// Mitsubishi GX Works2 project: PLC_GROUP13   PLC: FX3G

// global labels: Global1
VAR_GLOBAL
  StartDay AT X007 : BOOL;
END_VAR
VAR_GLOBAL CONSTANT
  input_choc : REAL := 1200;
END_VAR
VAR_GLOBAL
  chocStock AT D1152 : REAL;
END_VAR
VAR_GLOBAL CONSTANT
  input_nuts : REAL := 300;
END_VAR
VAR_GLOBAL
  nutsStock AT D1156 : REAL;
END_VAR
VAR_GLOBAL CONSTANT
  input_pist : REAL := 300;
END_VAR
VAR_GLOBAL
  pistStock AT D1160 : REAL;
END_VAR
VAR_GLOBAL CONSTANT
  input_kad : REAL := 120;
END_VAR
VAR_GLOBAL
  kadStock AT D1164 : REAL;
  melt AT X001 : BOOL;
END_VAR
VAR_GLOBAL CONSTANT
  subChoc : REAL := 400;
END_VAR
VAR_GLOBAL
  meltPot AT D1166 : REAL;
END_VAR
VAR_GLOBAL CONSTANT
  meltAdd : REAL := 400;
END_VAR
VAR_GLOBAL
  meltingIndicator AT Y001 : BOOL;
  fillStock AT M7 : BOOL;
END_VAR
VAR_GLOBAL CONSTANT
  minChoc : REAL := 400;
  minNuts : REAL := 100;
  minPist : REAL := 120;
  minKad : REAL := 60;
END_VAR
VAR_GLOBAL
  startDayLamp AT Y007 : BOOL;
END_VAR
VAR_GLOBAL CONSTANT
  Degrees : INT := 45;
END_VAR
VAR_GLOBAL
  TC_0 AT TC0 : BOOL;
  TC_1 AT TC1 : BOOL;
  TS_1 AT TS1 : BOOL;
  meltingProcess AT Y001 : BOOL;
  meltingEnded AT M3 : BOOL;
END_VAR
VAR_GLOBAL CONSTANT
  fourTrays : INT := 4;
END_VAR
VAR_GLOBAL
  placeTrays AT CC3 : BOOL;
  enterTray AT X010 : BOOL;
  traysPlaced AT CS3 : BOOL;
END_VAR
VAR_GLOBAL CONSTANT
  meltePour : REAL := 400;
  fourSeconds : INT := 40;
END_VAR
VAR_GLOBAL
  TC_2 AT TC2 : BOOL;
  pouring AT TC3 : BOOL;
  pouringEnded AT M4 : BOOL;
  pourChoc AT TS3 : BOOL;
  hi AT TS3 : BOOL;
  pourProcess AT Y002 : BOOL;
END_VAR
VAR_GLOBAL CONSTANT
  meltedPour : REAL := 400;
END_VAR
VAR_GLOBAL
  meltedChocPoured AT M6 : BOOL;
  chocMoved AT M5 : BOOL;
  meltingTime AT TC2 : BOOL;
  meltedPoured AT M6 : BOOL;
  applyChocType AT X004 : BOOL;
  chocTypeInput AT D8280 : INT;
  chocTypeSelected AT M10 : BOOL;
END_VAR
VAR_GLOBAL CONSTANT
  minForNuts : REAL;
  maxForNuts : REAL := 2025;
  minForDubai : REAL := 2025;
  maxForDubai : REAL := 4030;
  notGood : REAL := 3920;
  chocTypeNum : REAL := 1;
  removeNutsForNuts : REAL := 100;
  removePistForNuts : REAL := 100;
  nutsForFill : REAL := 200;
END_VAR
VAR_GLOBAL
  nutsMixing AT D1168 : REAL;
END_VAR
VAR_GLOBAL CONSTANT
  fillForNuts : REAL := 200;
  removeNutsForDubai : REAL := 20;
  removePistForDubai : REAL := 120;
  removeKadForDubai : REAL := 60;
  fillForDubai : REAL := 200;
END_VAR
VAR_GLOBAL
  dubaiMixing AT D1170 : REAL;
  mixingPot AT D1168 : REAL;
  ingredientsPoured AT M8 : BOOL;
  flashingLamp AT M9 : BOOL;
END_VAR
VAR_GLOBAL CONSTANT
  flashing3 : REAL := 50;
  fiveSec : INT := 50;
END_VAR
VAR_GLOBAL
  lampY3 AT Y003 : BOOL;
  lampY4 AT Y004 : BOOL;
  wordToReal AT M10 : BOOL;
  chocType1 AT D8202 : REAL;
  chocSelected AT M11 : BOOL;
  flashingTimerFive AT TC6 : BOOL;
  flashTimerEnd AT TS6 : BOOL;
  finishFlashingIndicator AT M12 : BOOL;
  chocSelection AT D1172 : REAL;
END_VAR
VAR_GLOBAL CONSTANT
  nutsSelected1 : REAL := 1;
  dubaiBling : REAL := 2;
  dubaiBling1 : REAL := 2;
END_VAR
VAR_GLOBAL
  chocIdentified AT M13 : BOOL;
  m_20 AT M20 : BOOL;
  m_21 AT M21 : BOOL;
END_VAR
VAR_GLOBAL CONSTANT
  fillForNuts1 : REAL := 200;
END_VAR
VAR_GLOBAL
  w AT M30 : BOOL;
END_VAR
VAR_GLOBAL CONSTANT
  halfSec : INT := 5;
END_VAR
VAR_GLOBAL
  coolChoc AT X006 : BOOL;
  TC_6 AT TC6 : BOOL;
  TS_6 AT TS6 : BOOL;
  coolingLamp AT Y006 : BOOL;
  finishCoolingIndicator AT M13 : BOOL;
  packTray AT X000 : BOOL;
  Packing AT CC4 : BOOL;
  traysPacked AT D1174 : REAL;
END_VAR
VAR_GLOBAL CONSTANT
  oneTray : REAL := 1;
  threeSeconds : INT := 30;
END_VAR
VAR_GLOBAL
  TS_7 AT TS7 : BOOL;
  PackingStartedIndicator AT M14 : BOOL;
  fourTraysPacked AT D1176 : REAL;
END_VAR
VAR_GLOBAL CONSTANT
  onePack : REAL := 1;
END_VAR
VAR_GLOBAL
  iterationEnded AT M15 : BOOL;
  emergency AT X005 : BOOL;
END_VAR
VAR_GLOBAL CONSTANT
  DivideByTen : REAL := 10;
END_VAR
VAR_GLOBAL
  trayscountOutput AT D8282 : INT;
END_VAR
VAR_GLOBAL CONSTANT
  zeroValue : REAL;
END_VAR
VAR_GLOBAL
  emergencyLamp AT M16 : BOOL;
END_VAR
VAR_GLOBAL CONSTANT
  fiftynine : REAL := 59;
END_VAR
VAR_GLOBAL
  outofStockLamp AT M17 : BOOL;
  intkadstock AT D1178 : INT;
  output AT D8282 : INT;
END_VAR
VAR_GLOBAL CONSTANT
  fourhundred : INT := 400;
  fourTy : REAL := 40;
  zero : INT;
END_VAR
VAR_GLOBAL
  dontaddLamp AT M18 : BOOL;
END_VAR
VAR_GLOBAL CONSTANT
  false_0 : BOOL;
END_VAR
VAR_GLOBAL
  meltingTimerFinished AT TS2 : BOOL;
  SelectedNuts AT M20 : BOOL;
  SelectedDubai AT M21 : BOOL;
  flashingTimer4 AT TC4 : BOOL;
  flashingTimer5 AT TC5 : BOOL;
  flashing4finish AT TS4 : BOOL;
  flashing5finish AT TS5 : BOOL;
  coolingTimer AT TC7 : BOOL;
  coolingTimerFinish AT TS7 : BOOL;
  Packed4Trays AT CS4 : BOOL;
  packingLamp AT Y005 : BOOL;
  chocInput AT D1180 : REAL;
  nutsInput AT D1182 : REAL;
  pistInput AT D1184 : REAL;
  kadInput AT D1186 : REAL;
END_VAR

// task Task_01 (event TRUE, interval 0, priority 31): POU_01

PROGRAM POU_01
VAR CONSTANT
  threeSec : INT := 30;
END_VAR
(* structured ladder/FBD written out as ST: instructions are called as NAME(EN, inputs, outputs); _pN, _eN, _tN stand for wires *)
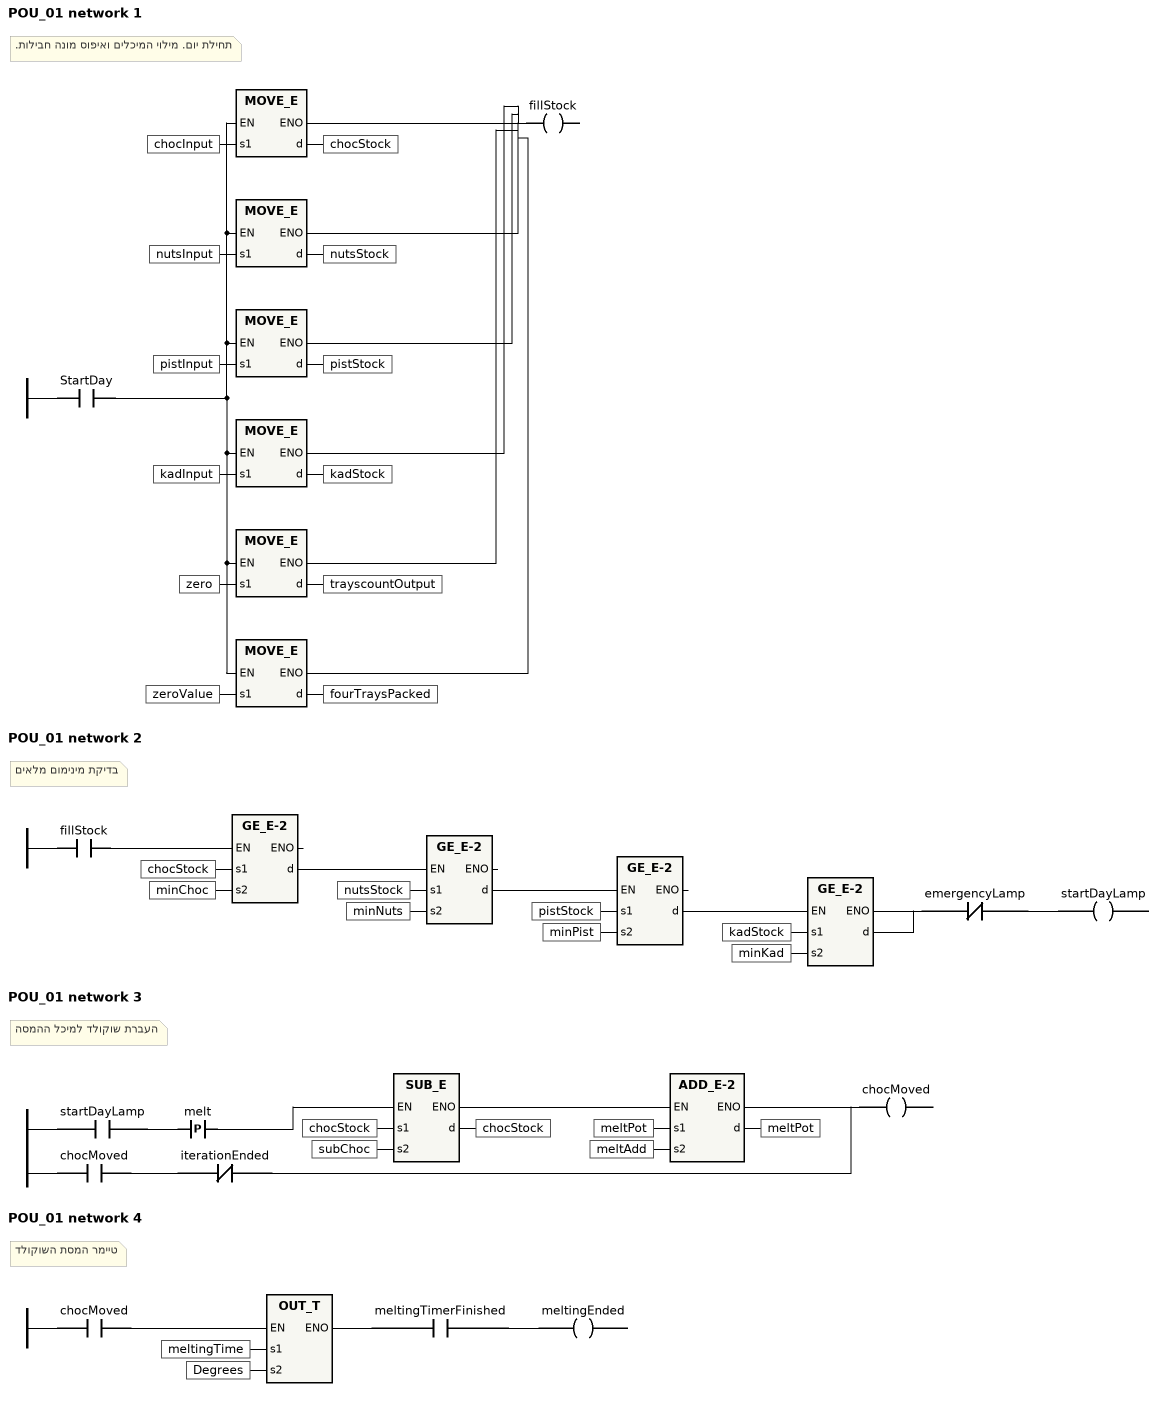
(* network 1 *)
(* תחילת יום. מילוי המיכלים ואיפוס מונה חבילות. *)
_e1 := MOVE_E(StartDay, chocInput, chocStock);
_e2 := MOVE_E(StartDay, nutsInput, nutsStock);
_e3 := MOVE_E(StartDay, pistInput, pistStock);
_e4 := MOVE_E(StartDay, kadInput, kadStock);
_e5 := MOVE_E(StartDay, zero, trayscountOutput);
_e6 := MOVE_E(StartDay, zeroValue, fourTraysPacked);
fillStock := _e1 OR _e2 OR _e3 OR _e4 OR _e5 OR _e6;
(* network 2 *)
(* בדיקת מינימום מלאים *)
GE_E(fillStock, chocStock, minChoc, _t1);
GE_E(_t1, nutsStock, minNuts, _t2);
GE_E(_t2, pistStock, minPist, _t3);
_e5 := GE_E(_t3, kadStock, minKad, _t4);
startDayLamp := (_e5 OR _t4) AND NOT emergencyLamp;
(* network 3 *)
(* העברת שוקולד למיכל ההמסה *)
_e1 := SUB_E(startDayLamp AND LDP(TRUE, melt), chocStock, subChoc, chocStock);
_e2 := ADD_E(_e1, meltPot, meltAdd, meltPot);
chocMoved := _e2 OR (chocMoved AND NOT iterationEnded);
(* network 4 *)
(* טיימר המסת השוקולד *)
_e1 := OUT_T(chocMoved, meltingTime, Degrees);
meltingEnded := _e1 AND meltingTimerFinished;
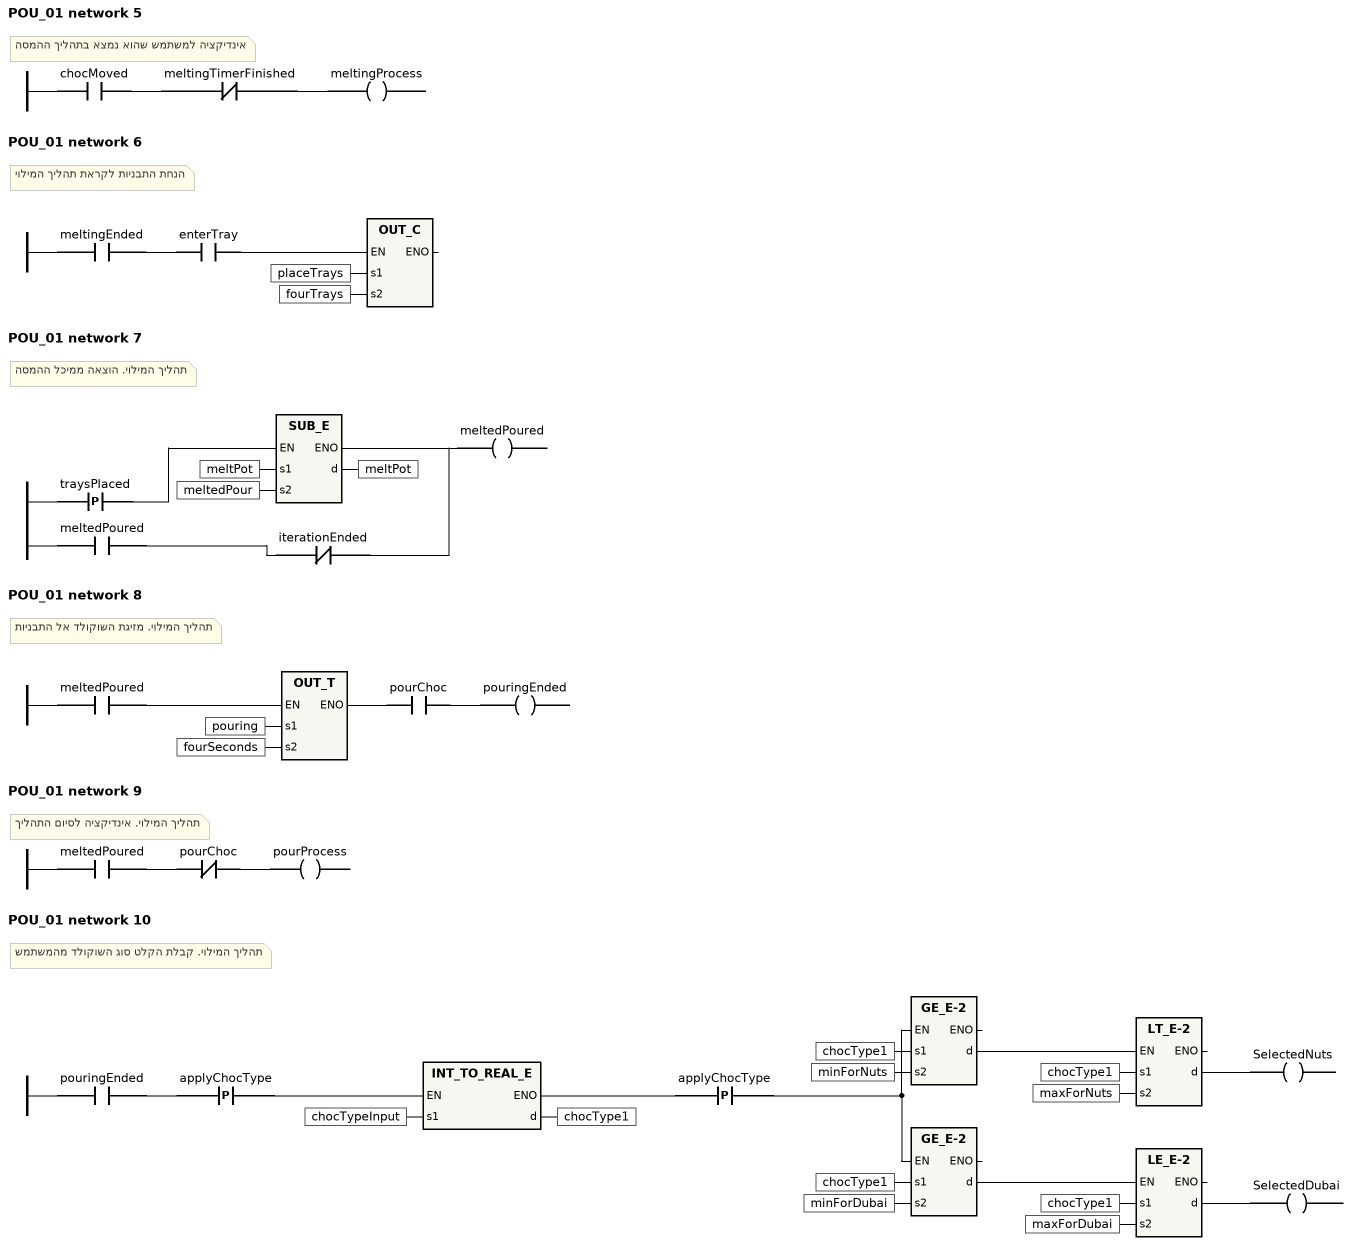
(* network 5 *)
(* אינדיקציה למשתמש שהוא נמצא בתהליך ההמסה *)
meltingProcess := chocMoved AND NOT meltingTimerFinished;
(* network 6 *)
(* הנחת התבניות לקראת תהליך המילוי *)
OUT_C(meltingEnded AND enterTray, placeTrays, fourTrays);
(* network 7 *)
(* תהליך המילוי. הוצאה ממיכל ההמסה *)
_e1 := SUB_E(LDP(TRUE, traysPlaced), meltPot, meltedPour, meltPot);
meltedPoured := _e1 OR (meltedPoured AND NOT iterationEnded);
(* network 8 *)
(* תהליך המילוי. מזיגת השוקולד אל התבניות *)
_e1 := OUT_T(meltedPoured, pouring, fourSeconds);
pouringEnded := _e1 AND pourChoc;
(* network 9 *)
(* תהליך המילוי. אינדיקציה לסיום התהליך *)
pourProcess := meltedPoured AND NOT pourChoc;
(* network 10 *)
(* תהליך המילוי. קבלת הקלט סוג השוקולד מהמשתמש *)
_e1 := INT_TO_REAL_E(pouringEnded AND LDP(TRUE, applyChocType), chocTypeInput, chocType1);
_p2 := _e1 AND LDP(TRUE, applyChocType);
GE_E(_p2, chocType1, minForNuts, _t3);
LT_E(_t3, chocType1, maxForNuts, _t4);
SelectedNuts := _t4;
GE_E(_p2, chocType1, minForDubai, _t5);
LE_E(_t5, chocType1, maxForDubai, _t6);
SelectedDubai := _t6;
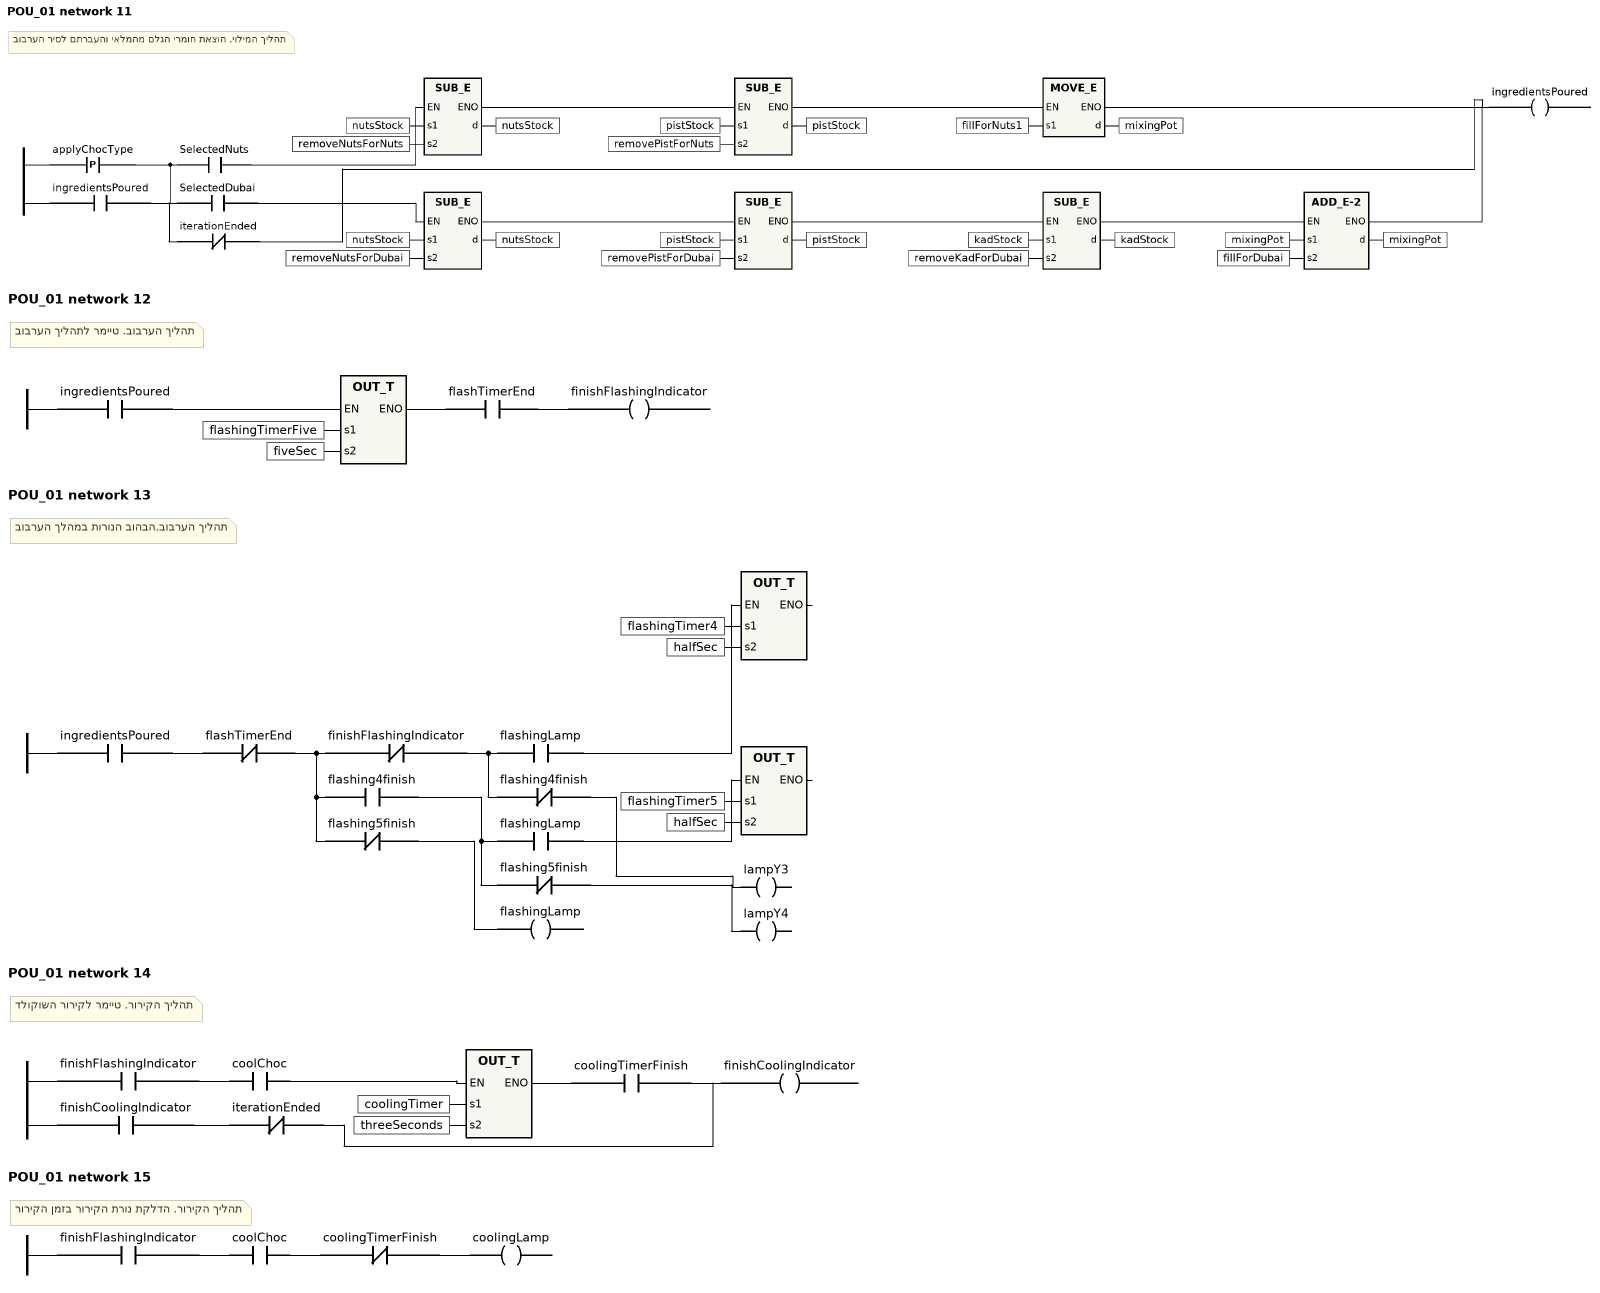
(* network 11 *)
(* תהליך המילוי. הוצאת חומרי הגלם מהמלאי והעברתם לסיר הערבוב *)
_p1 := LDP(TRUE, applyChocType);
_e2 := SUB_E(_p1 AND SelectedNuts, nutsStock, removeNutsForNuts, nutsStock);
_e3 := SUB_E(_e2, pistStock, removePistForNuts, pistStock);
_e4 := MOVE_E(_e3, fillForNuts1, mixingPot);
_e5 := SUB_E(_p1 AND SelectedDubai, nutsStock, removeNutsForDubai, nutsStock);
_e6 := SUB_E(_e5, pistStock, removePistForDubai, pistStock);
_e7 := SUB_E(_e6, kadStock, removeKadForDubai, kadStock);
_e8 := ADD_E(_e7, mixingPot, fillForDubai, mixingPot);
ingredientsPoured := _e4 OR _e8 OR (ingredientsPoured AND NOT iterationEnded);
(* network 12 *)
(* תהליך הערבוב. טיימר לתהליך הערבוב *)
_e1 := OUT_T(ingredientsPoured, flashingTimerFive, fiveSec);
finishFlashingIndicator := _e1 AND flashTimerEnd;
(* network 13 *)
(* תהליך הערבוב.הבהוב הנורות במהלך הערבוב *)
_p1 := ingredientsPoured AND NOT flashTimerEnd;
_p2 := _p1 AND NOT finishFlashingIndicator;
OUT_T(_p2 AND flashingLamp, flashingTimer4, halfSec);
lampY3 := _p2 AND NOT flashing4finish;
_p3 := _p1 AND flashing4finish;
OUT_T(_p3 AND flashingLamp, flashingTimer5, halfSec);
lampY4 := _p3 AND NOT flashing5finish;
flashingLamp := _p1 AND NOT flashing5finish;
(* network 14 *)
(* תהליך הקירור. טיימר לקירור השוקולד *)
_e1 := OUT_T(finishFlashingIndicator AND coolChoc, coolingTimer, threeSeconds);
finishCoolingIndicator := (_e1 AND coolingTimerFinish) OR (finishCoolingIndicator AND NOT iterationEnded);
(* network 15 *)
(* תהליך הקירור. הדלקת נורת הקירור בזמן הקירור *)
coolingLamp := finishFlashingIndicator AND coolChoc AND NOT coolingTimerFinish;
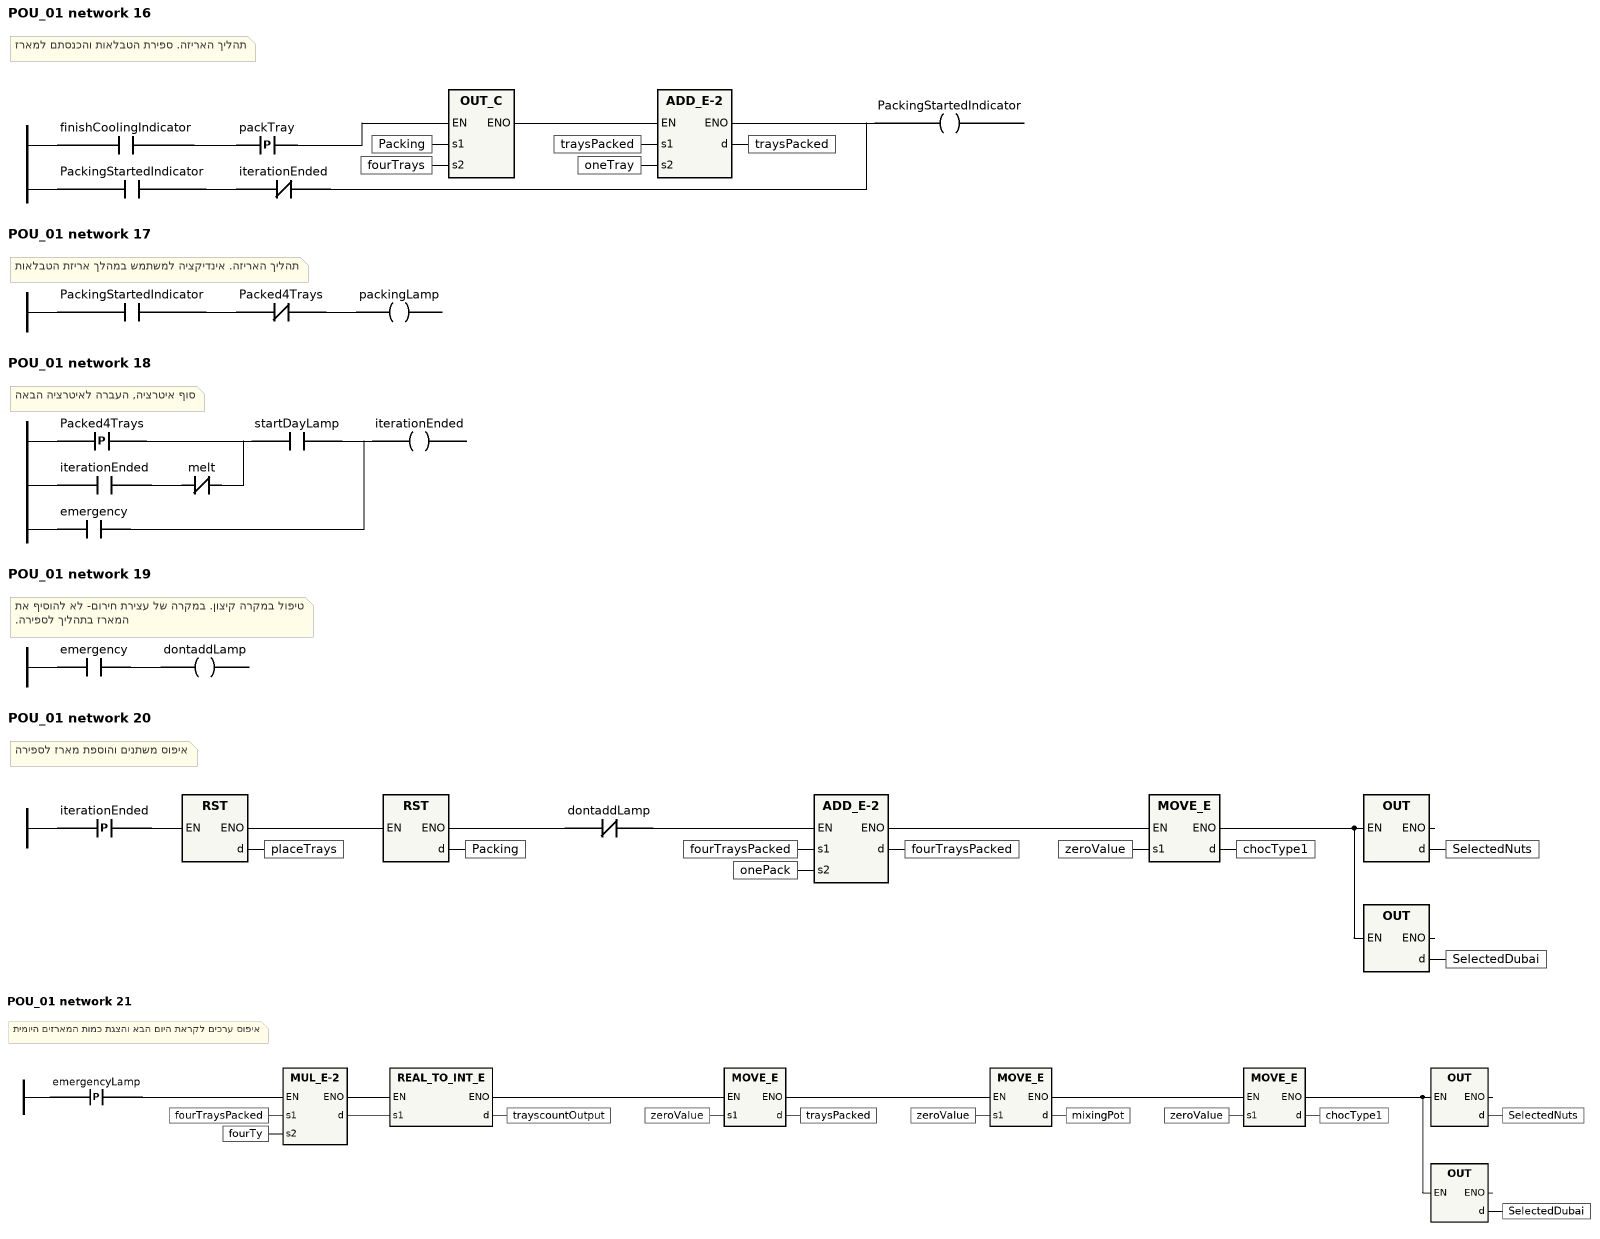
(* network 16 *)
(* תהליך האריזה. ספירת הטבלאות והכנסתם למארז *)
_e1 := OUT_C(finishCoolingIndicator AND LDP(TRUE, packTray), Packing, fourTrays);
_e2 := ADD_E(_e1, traysPacked, oneTray, traysPacked);
PackingStartedIndicator := _e2 OR (PackingStartedIndicator AND NOT iterationEnded);
(* network 17 *)
(* תהליך האריזה. אינדיקציה למשתמש במהלך אריזת הטבלאות *)
packingLamp := PackingStartedIndicator AND NOT Packed4Trays;
(* network 18 *)
(* סוף איטרציה, העברה לאיטרציה הבאה *)
iterationEnded := ((LDP(TRUE, Packed4Trays) OR (iterationEnded AND NOT melt)) AND startDayLamp) OR emergency;
(* network 19 *)
(* טיפול במקרה קיצון. במקרה של עצירת חירום- לא להוסיף את המארז בתהליך לספירה. *)
dontaddLamp := emergency;
(* network 20 *)
(* איפוס משתנים והוספת מארז לספירה *)
_e1 := RST(LDP(TRUE, iterationEnded), placeTrays);
_e2 := RST(_e1, Packing);
_e3 := ADD_E(_e2 AND NOT dontaddLamp, fourTraysPacked, onePack, fourTraysPacked);
_e4 := MOVE_E(_e3, zeroValue, chocType1);
OUT(_e4, SelectedNuts);
OUT(_e4, SelectedDubai);
(* network 21 *)
(* איפוס ערכים לקראת היום הבא והצגת כמות המארזים היומית *)
_e2 := MUL_E(LDP(TRUE, emergencyLamp), fourTraysPacked, fourTy, _t1);
_e3 := REAL_TO_INT_E(_e2, _t1, trayscountOutput);
_e4 := MOVE_E(_e3, zeroValue, traysPacked);
_e5 := MOVE_E(_e4, zeroValue, mixingPot);
_e6 := MOVE_E(_e5, zeroValue, chocType1);
OUT(_e6, SelectedNuts);
OUT(_e6, SelectedDubai);
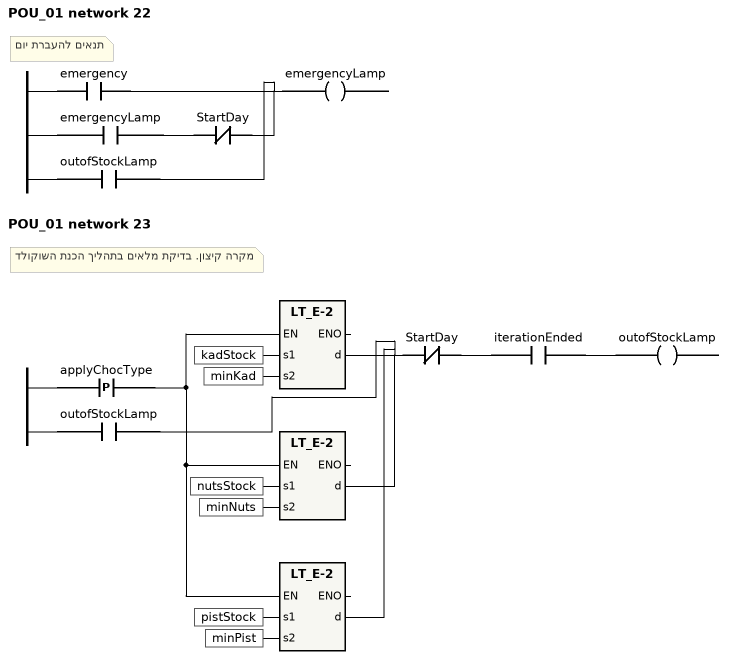
(* network 22 *)
(* תנאים להעברת יום *)
emergencyLamp := emergency OR (emergencyLamp AND NOT StartDay) OR outofStockLamp;
(* network 23 *)
(* מקרה קיצון. בדיקת מלאים בתהליך הכנת השוקולד *)
_p1 := LDP(TRUE, applyChocType);
LT_E(_p1, kadStock, minKad, _t2);
LT_E(_p1, nutsStock, minNuts, _t3);
LT_E(_p1, pistStock, minPist, _t4);
outofStockLamp := ((_t2 OR _t3 OR _t4 OR outofStockLamp) AND NOT StartDay) AND iterationEnded;
END_PROGRAM
